FUNCTION_BLOCK FB_SorterLogic (* Logique sorter - SIMPLIFIE *)
  (* Standard: 61499-2 *)
  (* Version 1.0, 20/01/2026, Claude, Schneider Electric, Version simplifiee *)
  PACKAGE Main;
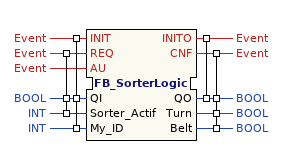
  EVENT_INPUT
    INIT WITH QI, My_ID; (* Initialization Request *)
    REQ WITH QI, Sorter_Actif; (* Normal Execution Request *)
    AU; (* Arret urgence *)
  END_EVENT
  EVENT_OUTPUT
    INITO WITH QO; (* Initialization Confirm *)
    CNF WITH QO, Turn, Belt; (* Execution Confirmation *)
  END_EVENT
  VAR_INPUT
    QI : BOOL; (* Input event qualifier *)
    Sorter_Actif : INT; (* ID du sorter actif *)
    My_ID : INT; (* Mon ID (1, 2 ou 3) *)
  END_VAR
  VAR_OUTPUT
    QO : BOOL; (* Output event qualifier *)
    Turn : BOOL; (* Tourner *)
    Belt : BOOL; (* Tapis *)
  END_VAR
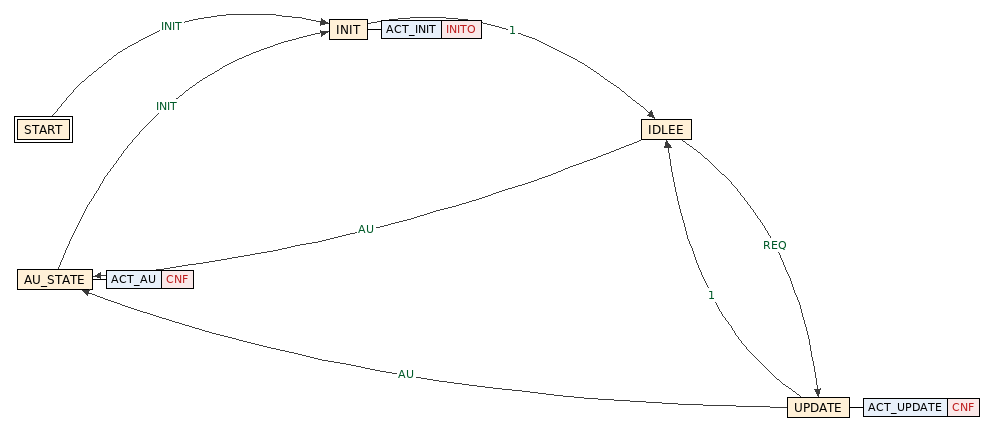
  EC_STATES
    START; (* Initial State *)
    INIT : ACT_INIT -> INITO; (* Initialization *)
    IDLEE; (* En attente *)
    UPDATE : ACT_UPDATE -> CNF; (* Mise a jour *)
    AU_STATE : ACT_AU -> CNF; (* Arret urgence *)
  END_STATES
  EC_TRANSITIONS
    START TO INIT := INIT;
    INIT TO IDLEE := 1;
    IDLEE TO UPDATE := REQ;
    UPDATE TO IDLEE := 1;
    IDLEE TO AU_STATE := AU;
    UPDATE TO AU_STATE := AU;
    AU_STATE TO INIT := INIT;
  END_TRANSITIONS
  ALGORITHM ACT_INIT IN ST: (* Initialization *)
QO := TRUE;
Turn := FALSE;
Belt := FALSE;
  END_ALGORITHM
  ALGORITHM ACT_UPDATE IN ST: (* Mise a jour sorter *)
(* Activer si c'est mon tour *)
IF Sorter_Actif = My_ID THEN
    Turn := TRUE;
    Belt := TRUE;
ELSE
    Turn := FALSE;
    Belt := FALSE;
END_IF;
  END_ALGORITHM
  ALGORITHM ACT_AU IN ST: (* Arret urgence *)
(* Tout arreter *)
Turn := FALSE;
Belt := FALSE;
  END_ALGORITHM
END_FUNCTION_BLOCK
